GVL_HMI.bVisionImagePrepared := fbVisionManualImages.bPrepared;
GVL_HMI.bVisionImage1Allowed := bVisionPbupKnown AND NOT bVisionPbupFitted;
IF NOT GVL_HMI.bVisionImage1Allowed AND (GVL_HMI.udiCameraManualImageSelection = 1) THEN
    GVL_HMI.udiCameraManualImageSelection := 0;
END_IF
GVL_HMI.bVisionPbupFittedApplied := bVisionPbupFitted;
GVL_HMI.bVisionPbupReferenceKnown := bVisionPbupKnown;
GVL_HMI.uiVisionPbupNest := uiVisionPbupNest;
GVL_HMI.bVisionImagePrepareAllowed := bVisionImagePermit AND bVisionPbupKnown
    AND NOT fbVisionManualImages.bBusy AND NOT fbVisionManualImages.bFault
    AND (usiManualCameraStep = 0)
    AND (fbVisionManualImages.bActive OR stVisionStatus.bHome)
    AND NOT GVL_HMI.bCameraManualBusy AND GVL_HMI.bCameraConnected
    AND GVL_EtherCAT.stVSKeyenceCamera.bRunStatus
    AND (GVL_HMI.udiCameraManualImageSelection >= 1) AND (GVL_HMI.udiCameraManualImageSelection <= 4)
    AND ((GVL_HMI.udiCameraManualImageSelection <> 1) OR NOT bVisionPbupFitted);
GVL_HMI.bVisionImageReleaseAllowed := fbVisionManualImages.bPrepared
    AND NOT fbVisionManualImages.bPartHeld AND (usiManualCameraStep = 0);
GVL_HMI.bCameraManualReady := bManualCameraTransportReady AND fbVisionManualImages.bPrepared
    AND (GVL_HMI.udiCameraManualImageSelection = fbVisionManualImages.udiPreparedImage)
    AND bVisionPbupKnown AND ((GVL_HMI.udiCameraManualImageSelection <> 1) OR NOT bVisionPbupFitted);
GVL_HMI.bCameraManualReady := GVL_HMI.bCameraManualReady
    OR (bManualCameraRecoveryAllowed AND NOT bManualCameraRecoveryActive);
GVL_HMI.bCameraManualBusy := GVL_HMI.bCameraManualBusy OR fbVisionManualImages.bBusy;
IF fbVisionManualImages.bActive OR fbVisionManualImages.bFault
    OR ((eMachineState = E_MachineState.Manual) AND stCommand.bVisionManualEnable) THEN
    GVL_HMI.sCameraManualMessage := fbVisionManualImages.sMessage;
END_IF
// One actionable reason. Prepared geometry is independent of camera transport.
IF (eMachineState = E_MachineState.Manual) AND stCommand.bVisionManualEnable THEN
    IF NOT stInputs.stSafety.bSafetyOk THEN
        GVL_HMI.sCameraManualMessage := 'Vision blocked: safety not ready';
    ELSIF NOT stInputs.bMainDoorClosed OR NOT GVL_Safety.bAirSupplySafe THEN
        GVL_HMI.sCameraManualMessage := 'Vision blocked: close door / restore air';
    ELSIF bManualCameraRecoveryActive OR bManualCameraRecoveryFailed THEN
        GVL_HMI.sCameraManualMessage := sManualCameraRecoveryMessage;
    ELSIF fbVisionManualImages.bCameraWarning AND fbVisionManualImages.bBusy THEN
        GVL_HMI.sCameraManualMessage := fbVisionManualImages.sMessage;
    ELSIF bVisionCameraStartBlocked THEN
        GVL_HMI.sCameraManualMessage := 'Camera error - use Camera Reset or retry Trigger';
    ELSIF NOT GVL_HMI.bCameraConnected OR NOT GVL_EtherCAT.stVSKeyenceCamera.bRunStatus THEN
        GVL_HMI.sCameraManualMessage := 'Camera not connected / not in RUN';
    ELSIF stIndexStatus.bBusy OR stIndexStatus.bTwoHandRequired
        OR (stInputs.bTwoHandsSafe AND NOT fbVisionManualImages.bActive)
        OR NOT stInputs.bIndexReady OR NOT stInputs.bIndexLocked
        OR (stInputs.eIndexPosition = E_TablePosition.Unknown) THEN
        GVL_HMI.sCameraManualMessage := 'Wait for locked index; release two-hand';
    ELSIF bRejectChuteStopRequestLatched OR stCommand.bStop OR stCommand.bReset THEN
        GVL_HMI.sCameraManualMessage := 'Vision blocked: Stop/Reset active';
    ELSIF NOT stVisionNest.bPartPresent THEN
        GVL_HMI.sCameraManualMessage := 'No tracked product at Vision';
    ELSIF fbVisionManualImages.bFault OR fbVisionManualImages.bBusy THEN
        GVL_HMI.sCameraManualMessage := fbVisionManualImages.sMessage;
    ELSIF bVisionImageJogBusy OR bVisionManualSequenceActive OR bVisionManualHomeActive THEN
        GVL_HMI.sCameraManualMessage := 'Finish Vision jog / HOME / sequence first';
    ELSIF fbVisionManualImages.bCameraWarning THEN
        GVL_HMI.sCameraManualMessage := fbVisionManualImages.sMessage;
    ELSIF NOT bVisionPbupKnown THEN
        GVL_HMI.sCameraManualMessage := 'Confirm PBUP fitted state for this nest';
    ELSIF (GVL_HMI.udiCameraManualImageSelection < 1) OR (GVL_HMI.udiCameraManualImageSelection > 4) THEN
        GVL_HMI.sCameraManualMessage := 'Select an image';
    ELSIF (GVL_HMI.udiCameraManualImageSelection <> 1) AND NOT bVisionPbupFitted
        AND NOT stVisionNest.bLoadSetComplete THEN
        GVL_HMI.sCameraManualMessage := 'Mounting requires a complete paired load';
    ELSIF NOT fbVisionManualImages.bActive AND NOT stVisionStatus.bHome THEN
        GVL_HMI.sCameraManualMessage := 'Return Vision tooling HOME before Prepare';
    ELSIF bManualCameraDrainResult THEN
        GVL_HMI.sCameraManualMessage := 'Camera: clearing previous result handshake';
    ELSIF GVL_HMI.bCameraManualBusy THEN
        GVL_HMI.sCameraManualMessage := 'Camera: loading program / capture in progress';
    ELSIF fbVisionManualImages.bPrepared
        AND (GVL_HMI.udiCameraManualImageSelection = fbVisionManualImages.udiPreparedImage) THEN
        IF bManualCameraTransportReady THEN
            GVL_HMI.sCameraManualMessage := 'Position ready - press Camera Trigger';
        ELSE
            GVL_HMI.sCameraManualMessage := 'Position ready - waiting for camera handshake';
        END_IF
    ELSE
        GVL_HMI.sCameraManualMessage := 'Press Prepare Position for the selected image';
    END_IF
END_IF
GVL_HMI.sVisionPbupStatus := CONCAT('Nest ', UINT_TO_STRING(uiVisionPbupNest));
IF (uiVisionPbupNest < 1) OR (uiVisionPbupNest > 4) THEN
    GVL_HMI.sVisionPbupStatus := 'Wait for a known, locked index position';
ELSIF NOT stVisionNest.bPartPresent THEN
    GVL_HMI.sVisionPbupStatus := CONCAT(GVL_HMI.sVisionPbupStatus, ': no tracked part; load at operator station');
ELSIF NOT bVisionPbupKnown THEN
    GVL_HMI.sVisionPbupStatus := CONCAT(GVL_HMI.sVisionPbupStatus, ': confirm saved PBUP state');
ELSIF bVisionPbupFitted THEN
    GVL_HMI.sVisionPbupStatus := CONCAT(GVL_HMI.sVisionPbupStatus, ': PBUP fitted');
ELSE
    GVL_HMI.sVisionPbupStatus := CONCAT(GVL_HMI.sVisionPbupStatus, ': PBUP not fitted');
END_IF
IF stVisionNest.bPartPresent AND bVisionPbupKnown AND (uiVisionPbupNest >= 1) AND (uiVisionPbupNest <= 4) THEN
    IF aVisionPbupSource[uiVisionPbupNest] = 1 THEN
        GVL_HMI.sVisionPbupStatus := CONCAT(GVL_HMI.sVisionPbupStatus, ' / new paired load');
    ELSIF aVisionPbupSource[uiVisionPbupNest] = 2 THEN
        GVL_HMI.sVisionPbupStatus := CONCAT(GVL_HMI.sVisionPbupStatus, ' / operator confirmed');
    ELSE
        GVL_HMI.sVisionPbupStatus := CONCAT(GVL_HMI.sVisionPbupStatus, ' / mounting completed');
    END_IF
END_IF


// Native event grid is the single engineer-feedback presentation on this tab.
GVL_MASTER.bVisionManualCameraWarning := (eMachineState = E_MachineState.Manual)
    AND fbVisionManualImages.bCameraWarning;
GVL_MASTER.bVisionManualGridActive := (eMachineState = E_MachineState.Manual)
    AND stCommand.bVisionManualEnable;
GVL_MASTER.bVisionManualGridWarning := GVL_MASTER.bVisionManualGridActive
    AND NOT GVL_HMI.bCameraManualReady AND NOT GVL_HMI.bCameraManualBusy
    AND NOT fbVisionManualImages.bFault AND NOT fbVisionManualImages.bCameraWarning
    AND NOT bVisionCameraStartBlocked AND NOT bManualCameraRecoveryFailed;

// =====================================================
// VISION MANUAL MODE - HOME COMPLETION
// =====================================================

// Release Home ownership once FB_VisionStation has
// completed the controlled homing sequence and is Ready.
IF (eMachineState = E_MachineState.Manual)
    AND bVisionManualHomeActive
    AND fbVision.IsReady()
THEN
    bVisionManualHomeActive := FALSE;
END_IF;

// Release Home ownership if Vision enters Fault.
IF (eMachineState = E_MachineState.Manual)
    AND bVisionManualHomeActive
    AND fbVision.IsFaulted()
THEN
    bVisionManualHomeActive := FALSE;
END_IF;

// =====================================================
// VISION MANUAL MODE - RUN SEQUENCE COMPLETION
// =====================================================

// Complete manual Run Sequence.
// Return FB_VisionStation from Done to Ready.
IF (eMachineState = E_MachineState.Manual)
    AND bVisionManualSequenceActive
    AND fbVision.IsDone()
THEN
    fbVision.RequestReset();
    bVisionManualSequenceActive := FALSE;
END_IF;


// Abort manual Run Sequence ownership if Vision faults.
// The station fault remains available for the normal
// machine fault / diagnostic handling.
IF (eMachineState = E_MachineState.Manual)
    AND bVisionManualSequenceActive
    AND fbVision.IsFaulted()
THEN
    bVisionManualSequenceActive := FALSE;
END_IF;
// =====================================================
// VISION MANUAL MODE - OUTPUT OVERRIDE
// =====================================================
// Applied AFTER fbVision.Update() because FB_VisionStation owns these
// requests during Initialising / ReadyToStart / AutoCycle.
//
// Manual movement is accepted only when:
//   Manual Mode + Safety OK + Vision Manual Enable + movement permissive.
//
// Opposite requests are mutually interlocked here in the PLC.

// If Vision manual control is not enabled/allowed, do not permit any manual
// Vision motion request to survive into the physical output image.
IF (eMachineState = E_MachineState.Manual)
    AND NOT bVisionManualSequenceActive
    AND NOT bVisionManualHomeActive
    AND NOT fbVisionManualImages.bActive AND NOT bVisionImageOwnedBeforeUpdate
    AND NOT fbVisionManualImages.bFault
THEN

    // Start from a safe manual command image every scan.
    bVisionHorizontalBackRequest := FALSE;
    bVisionHorizontalFrontRequest := FALSE;
    bVisionVerticalUpRequest := FALSE;
    bVisionVerticalDownRequest := FALSE;

    bVisionGripCloseRequest := FALSE;
    bVisionGripOpenRequest := FALSE;
    bVisionRotate0Request := FALSE;
    bVisionRotate180Request := FALSE;



    // =====================================================
    // VISION MANUAL - COMMAND EDGES
    // =====================================================

    // Horizontal - KEEP EXACTLY AS VALIDATED
    rtVisionManualHorizontalBack(
        CLK := stCommand.bVisionHorizontalBackRequest
    );

    rtVisionManualHorizontalFront(
        CLK := stCommand.bVisionHorizontalFrontRequest
    );

//     // Vertical
//     rtVisionManualVerticalUp(
//         CLK := stCommand.bVisionVerticalUpRequest
//     );
// 
//     );
// 
//     rtVisionManualVerticalFullDown(
//         CLK := stCommand.bVisionVerticalFullDownRequest
//     );
// 
// 	rtVisionManualGripOpen(
// 		CLK := stCommand.bVisionGripOpenRequest
// 	);
// 	
// 	rtVisionManualGripClose(
// 		CLK := stCommand.bVisionGripCloseRequest
// 	);

    IF bVisionManualEnableAllowed
        AND stCommand.bVisionManualEnable
    THEN


        // =====================================================
        // VISION MANUAL - HORIZONTAL
        // =====================================================
        // KEEP EXACTLY AS VALIDATED.
        //
        // BACK = HOME

        tpVisionManualHorizontalBack(
            IN :=
                rtVisionManualHorizontalBack.Q
                AND bVisionHorizontalBackAllowed,
            PT := T#1S
        );

        // FRONT
        tpVisionManualHorizontalFront(
            IN :=
                rtVisionManualHorizontalFront.Q
                AND bVisionHorizontalFrontAllowed,
            PT := T#1S
        );

	

        // Never command both directions simultaneously.
        IF tpVisionManualHorizontalBack.Q
            AND NOT tpVisionManualHorizontalFront.Q
        THEN

            bVisionHorizontalBackRequest := TRUE;
            bVisionHorizontalFrontRequest := FALSE;

        ELSIF tpVisionManualHorizontalFront.Q
            AND NOT tpVisionManualHorizontalBack.Q
        THEN

            bVisionHorizontalFrontRequest := TRUE;
            bVisionHorizontalBackRequest := FALSE;

        END_IF;

		// =====================================================
		// VISION MANUAL - VERTICAL
		// =====================================================
		//
		// UP:
		//     Vertical UP until UP feedback.
		//
		// INTERMEDIATE:
		//     3. Drive Vertical DOWN.
		//     4. Stop command when cylinder leaves UP.
		//
		// FULL DOWN:
		//     3. Drive Vertical DOWN.
		//     4. Stop at full DOWN feedback.
		//
		// HMI commands are one-scan requests.
		// No timer is used.
		
		
		// -----------------------------------------------------
		// ACCEPT NEW TARGET
		// -----------------------------------------------------
		
        IF stCommand.bVisionVerticalUpRequest AND bVisionVerticalUpAllowed THEN
            bVisionManualVerticalUpActive := TRUE;
            bVisionManualVerticalFullDownActive := FALSE;
        ELSIF stCommand.bVisionVerticalFullDownRequest AND bVisionVerticalFullDownAllowed THEN
            bVisionManualVerticalUpActive := FALSE;
            bVisionManualVerticalFullDownActive := TRUE;
        END_IF
        IF bVisionManualVerticalUpActive THEN
            bVisionVerticalDownRequest := FALSE;
            bVisionVerticalUpRequest := NOT stInputs.bVerticalMiniSlideRetracted;
            IF stInputs.bVerticalMiniSlideRetracted THEN
                bVisionVerticalUpRequest := FALSE;
                bVisionManualVerticalUpActive := FALSE;
            END_IF
        ELSIF bVisionManualVerticalFullDownActive THEN
            bVisionVerticalUpRequest := FALSE;
            bVisionVerticalDownRequest := NOT stInputs.bVerticalMiniSlideExtended;
            IF stInputs.bVerticalMiniSlideExtended THEN
                bVisionVerticalDownRequest := FALSE;
                bVisionManualVerticalFullDownActive := FALSE;
            END_IF
        END_IF

		// =====================================================
		// VISION MANUAL - GRIP
		// =====================================================
		// Momentary command.
		// HMI request is converted to a one-scan PLC pulse in
		// PRG_HmiCommands.
		//
		// No timer is required.
		// OPEN and CLOSE are mutually exclusive.
		
		IF stCommand.bVisionGripOpenRequest
			AND NOT stCommand.bVisionGripCloseRequest
			AND bVisionGripOpenAllowed
		THEN
		
			bVisionGripOpenRequest := TRUE;
			bVisionGripCloseRequest := FALSE;
		
		ELSIF stCommand.bVisionGripCloseRequest
			AND NOT stCommand.bVisionGripOpenRequest
			AND bVisionGripCloseAllowed
		THEN
		
			bVisionGripOpenRequest := FALSE;
			bVisionGripCloseRequest := TRUE;
		
		ELSE
		
			bVisionGripOpenRequest := FALSE;
			bVisionGripCloseRequest := FALSE;
		
		END_IF


		// =====================================================
		// VISION MANUAL - ROTATION
		// =====================================================
		// HMI command is a one-scan request.
		// PLC keeps the output active until position feedback.
		// No timer is required.
		
		// Start 0Â°
		IF stCommand.bVisionRotate0Request
			AND bVisionRotate0Allowed
			AND NOT bVisionManualRotate180Active
		THEN
			bVisionManualRotate0Active := TRUE;
		END_IF
		
		// Start 180Â°
		IF stCommand.bVisionRotate180Request
			AND bVisionRotate180Allowed
			AND NOT bVisionManualRotate0Active
		THEN
			bVisionManualRotate180Active := TRUE;
		END_IF
		
		// Execute movement
		IF bVisionManualRotate0Active THEN
		
			bVisionRotate0Request := TRUE;
			bVisionRotate180Request := FALSE;
		
			IF bVisionRotate0Confirmed THEN
				bVisionRotate0Request := FALSE;
				bVisionManualRotate0Active := FALSE;
			END_IF
		
		ELSIF bVisionManualRotate180Active THEN
		
			bVisionRotate0Request := FALSE;
			bVisionRotate180Request := TRUE;
		
			IF bVisionRotate180Confirmed THEN
				bVisionRotate180Request := FALSE;
				bVisionManualRotate180Active := FALSE;
			END_IF
		
		ELSE
		
			bVisionRotate0Request := FALSE;
			bVisionRotate180Request := FALSE;
		
		END_IF


	ELSE
	
		// Vision Manual Enable removed:
		// cancel unfinished manual movements.

		bVisionManualVerticalUpActive := FALSE;
		bVisionManualVerticalFullDownActive := FALSE;
		bVisionManualRotate0Active := FALSE;
		bVisionManualRotate180Active := FALSE;
	
	END_IF

ELSE

    // Leaving Manual also cancels unfinished manual sequences.
    bVisionManualVerticalUpActive := FALSE;

    bVisionManualVerticalFullDownActive := FALSE;

    bVisionManualRotate0Active := FALSE;
    bVisionManualRotate180Active := FALSE;

END_IF

stVisionStatus.bFault := stVisionStatus.bFault OR fbVisionManualImages.bFault;
IF fbVisionManualImages.bActive OR fbVisionManualImages.bFault THEN
    stVisionStatus.sDiagnostic := fbVisionManualImages.sMessage;
END_IF

// Current station/nest status for HMI.
stPatchDispenseStatus.bPartPresent := bPatchDispenseRequired;
stHeatStakeStatus.bPartPresent := bHeatStakeRequired;
stVisionStatus.bPartPresent := bVisionRequired;

// Homing is an internal machine-initialisation activity, not an automatic
// process cycle. Keep FB_VisionStation.IsBusy() unchanged for controlled-stop
// logic, but do not publish Vision as Busy to the operator while the machine is
// in System Initialising.
IF eMachineState = E_MachineState.Initialising THEN
    stVisionStatus.bBusy := FALSE;
END_IF

// Manual indication follows current HOME feedback, independently of the station FB state.
// Individual manual movements are owned by the machine and can leave the station FB idle.
IF eMachineState = E_MachineState.Manual THEN
    stVisionStatus.bBusy :=
        NOT stVisionStatus.bHome
        OR bVisionManualSequenceActive
        OR bVisionManualHomeActive
        OR fbVisionManualImages.bActive;

    stVisionStatus.bReady :=
        stVisionStatus.bHome
        AND NOT stVisionStatus.bBusy
        AND bVisionManualEnableAllowed
        AND stCommand.bVisionManualEnable
        AND NOT fbVision.IsFaulted() AND NOT fbVisionManualImages.bFault;
END_IF

// "Ready" on the Heat Stake HMI is an operational indication, not an
// Initialising indication.
//
// FB_HeatStakeStation is intentionally enabled during System Initialising so
// it can establish/check its safe initial position. Its internal IsReady()
// state is still allowed to become TRUE there, because machine Initialising
// may depend on it. Only the published HMI Ready indication is gated.
//
// Show Ready only in states where an engineer/operator can actually use the
// station.
stHeatStakeStatus.bReady :=
    stHeatStakeStatus.bReady
    AND (
        (eMachineState = E_MachineState.ReadyToStart)
        OR (eMachineState = E_MachineState.AutoCycle)
        OR (eMachineState = E_MachineState.Manual)
    );

IF NOT bPatchDispenseRequired THEN
    stPatchDispenseStatus.eResultStatus := E_StationResultStatus.NotTested;
ELSIF stPatchDispenseNest.stPatchDispenseResult.bValid THEN
    IF stPatchDispenseNest.stPatchDispenseResult.bPassed THEN
        stPatchDispenseStatus.eResultStatus := E_StationResultStatus.Pass;
    ELSE
        stPatchDispenseStatus.eResultStatus := E_StationResultStatus.Fail;
    END_IF
ELSE
    stPatchDispenseStatus.eResultStatus := E_StationResultStatus.NotTested;
END_IF

IF stHeatStakeNest.stHeatStakeResult.bValid
    AND (stHeatStakeNest.stHeatStakeResult.udiAlertCode = GVL_MASTER.udiHeatStakePatchMissingAlertCode) THEN
    stHeatStakeStatus.eResultStatus := E_StationResultStatus.Fail;
ELSIF NOT bHeatStakeRequired THEN
    stHeatStakeStatus.eResultStatus := E_StationResultStatus.NotTested;
ELSIF stHeatStakeNest.stHeatStakeResult.bValid THEN
    IF stHeatStakeNest.stHeatStakeResult.bPassed THEN
        stHeatStakeStatus.eResultStatus := E_StationResultStatus.Pass;
    ELSE
        stHeatStakeStatus.eResultStatus := E_StationResultStatus.Fail;
    END_IF
ELSE
    stHeatStakeStatus.eResultStatus := E_StationResultStatus.NotTested;
END_IF

IF NOT bVisionRequired THEN
    stVisionStatus.eResultStatus := E_StationResultStatus.NotTested;
ELSIF stVisionNest.stVisionResult.bValid THEN
    IF stVisionNest.stVisionResult.bPassed THEN
        stVisionStatus.eResultStatus := E_StationResultStatus.Pass;
    ELSE
        stVisionStatus.eResultStatus := E_StationResultStatus.Fail;
    END_IF
ELSE
    stVisionStatus.eResultStatus := E_StationResultStatus.NotTested;
END_IF

bAllRequiredStationsReady :=
    ((NOT bPatchDispenseRequired) OR fbPatchDispense.IsReady())
    AND ((NOT bHeatStakeRequired) OR fbHeatStake.IsReady())
    AND ((NOT bVisionRequired) OR fbVision.IsReady());

bAllRequiredStationsComplete :=
    ((NOT bPatchDispenseRequired) OR fbPatchDispense.IsDone())
    AND ((NOT bHeatStakeRequired) OR fbHeatStake.IsDone())
    AND ((NOT bVisionRequired) OR fbVision.IsDone());

// TRUE from support extension through the simulated process and support
// retraction of at least one active station.
bAnyStationInProcess :=
    fbPatchDispense.IsBusy()
    OR fbHeatStake.IsBusy()
    OR fbVision.IsBusy();

IF (eProcessCycleState = E_CycleState.WaitingForProcessesComplete)
    AND bAllRequiredStationsComplete
    AND NOT bCycleResultsStored
THEN

	IF bPatchDispenseRequired THEN
	
		// Capture the station result once.
		stPatchDispenseCycleResult := fbPatchDispense.GetResult();
	
		// Store the Patch Dispense result in the physical nest.
		fbNestManager.StorePatchDispenseResultAtPosition(
			ePosition := stConfig.ePatchDispensePosition,
			stResult := stPatchDispenseCycleResult
		);
	
		IF stPatchDispenseCycleResult.bValid AND NOT stPatchDispenseCycleResult.bPassed THEN
			FinaliseAndRecordAtPosition(stConfig.ePatchDispensePosition);
		END_IF

	END_IF

    IF bHeatStakeRequired THEN
        stHeatStakeCycleResult := fbHeatStake.GetResult();
        fbNestManager.StoreHeatStakeResultAtPosition(
            ePosition := stConfig.eHeatStakePosition,
            stResult := stHeatStakeCycleResult
        );
        IF stHeatStakeCycleResult.bValid AND NOT stHeatStakeCycleResult.bPassed THEN
            FinaliseAndRecordAtPosition(stConfig.eHeatStakePosition);
        END_IF
    END_IF

    IF bVisionRequired THEN
        fbNestManager.StoreVisionResultAtPosition(
            ePosition := stConfig.eVisionPosition,
            stResult := fbVision.GetResult()
        );
    END_IF
	
    FinaliseAndRecordAtPosition(stConfig.eVisionPosition);

// Prevent this cycle result from being stored/finalised again.
bCycleResultsStored := TRUE;


END_IF

// =====================================================
// REPROCESS POPUP - OPERATOR STATION
// =====================================================
// 
// Activate Reprocess requirement when a Reprocess
// part is present at the Operator Station.
IF (stOperatorNest.ePosition = E_TablePosition.Position1)
    AND (stOperatorNest.eDisposition = E_PartDisposition.Reprocess)
    AND stOperatorNest.bPartPresent
THEN
    bReprocessAcknowledgePending := TRUE;
END_IF

// Reset acknowledgement memory only when there is
// no active Reprocess acknowledgement pending
// and the operator nest is empty.
IF NOT stOperatorNest.bPartPresent
    AND NOT bReprocessAcknowledgePending
THEN
    bReprocessPopupAcknowledged := FALSE;
END_IF

// Acknowledge the current Reprocess part.
IF GVL_HMI.stCommands.bReprocessPopupAcknowledge THEN
    bReprocessPopupAcknowledged := TRUE;
    bReprocessAcknowledgePending := FALSE;
    GVL_HMI.stCommands.bReprocessPopupAcknowledge := FALSE;
END_IF

// // Require acknowledgement only for an unacknowledged
// // Reprocess part physically present at the Operator Station.
// IF (stOperatorNest.ePosition = E_TablePosition.Position1)
//     AND (stOperatorNest.eDisposition = E_PartDisposition.Reprocess)
//     AND stOperatorNest.bPartPresent
//     AND NOT bReprocessPopupAcknowledged
// THEN
//     bReprocessAcknowledgePending := TRUE;
// END_IF

// Popup remains requested until acknowledged,
// // even if the part is physically removed.
// GVL_HMI.stStatus.bReprocessPopupRequest :=
//     bReprocessAcknowledgePending;
// Reprocess popup request.
// Keep the PLC interlock independent from popup visibility.

rtReprocessIndexAttempt(
    CLK := stInputs.bTwoHandsSafe
);

// Generate a new FALSE -> TRUE transition when the
// operator attempts to index with Reprocess pending.
IF NOT bReprocessAcknowledgePending THEN

    GVL_HMI.stStatus.bReprocessPopupRequest := FALSE;

ELSIF rtReprocessIndexAttempt.Q THEN

    GVL_HMI.stStatus.bReprocessPopupRequest := FALSE;

ELSE

    GVL_HMI.stStatus.bReprocessPopupRequest := TRUE;

END_IF
// Request popup only for an unacknowledged Reprocess part
// physically present at the Operator Station.
// GVL_HMI.stStatus.bReprocessPopupRequest :=
//     (stOperatorNest.ePosition = E_TablePosition.Position1)
//     AND (stOperatorNest.eDisposition = E_PartDisposition.Reprocess)
//     AND stOperatorNest.bPartPresent
//     AND NOT bReprocessPopupAcknowledged;

// Clear an old processed record only after operator disposition is complete.
// A newly loaded part is not cleared because its load edge has already reset
// stResult.bValid to FALSE in FB_NestTableManager.
IF stOperatorStatus.bExchangeComplete
    AND (
        stOperatorNest.stResult.bValid
        OR (stOperatorNest.eDisposition = E_PartDisposition.Reprocess)
    )
    AND NOT stInputs.bLoadingStationEaglePresent
    AND NOT stInputs.bLoadingStationPbupPresent
THEN

    fbNestManager.ClearOperatorNest(
        stConfig.eOperatorPosition
    );

END_IF




stOutputsInternal.bStation1SupportExtend := FALSE; // Removed Station 1 nest support.
stOutputsInternal.bStation1SupportRetract := FALSE; // Reserved compatibility output.
stOutputsInternal.bStation2SupportExtend := bStation2SupportExtendRequest;
stOutputsInternal.bStation2SupportRetract := bStation2SupportRetractRequest;
stOutputsInternal.bStation3SupportExtend := FALSE; // Removed hardware.
stOutputsInternal.bStation3SupportRetract := FALSE; // Removed hardware.
stOutputsInternal.bVisionHorizontalBack := bVisionHorizontalBackRequest;
stOutputsInternal.bVisionHorizontalFront := bVisionHorizontalFrontRequest;
stOutputsInternal.bVisionVerticalUp := bVisionVerticalUpRequest;
stOutputsInternal.bVisionVerticalDown := bVisionVerticalDownRequest;
stOutputsInternal.bVisionLimitOff := FALSE; // Removed hardware.
stOutputsInternal.bVisionLimitOn := FALSE; // Removed hardware.
stOutputsInternal.bVisionGripClose := bVisionGripCloseRequest;
stOutputsInternal.bVisionGripOpen := bVisionGripOpenRequest;
stOutputsInternal.bVisionRotate0 := bVisionRotate0Request;
stOutputsInternal.bVisionRotate180 := bVisionRotate180Request;
stOutputsInternal.bHeatStakeHeadLock := bHeatStakeHeadLockRequest;
stOutputsInternal.bHeatStakeHeadUnlock := bHeatStakeHeadUnlockRequest;
stOutputsInternal.bHeatStakeHeadDown := bHeatStakeHeadDownRequest;
stOutputsInternal.bHeatStakeHeadUp := bHeatStakeHeadUpRequest;
stPermissives.bAirSupplyReady := GVL_Safety.bAirSupplySafe;


// Patch actuator ownership: HOME/sequence, individual Manual actions, then index hold-UP.
bPatchHoldUpAllowed := bPatchDispenseCommissioned AND stInputs.stSafety.bSafetyOk
    AND stInputs.bMainDoorClosed AND GVL_Safety.bAirSupplySafe
    AND ((eMachineState = E_MachineState.AutoCycle)
        OR ((eMachineState = E_MachineState.Manual)
            AND NOT bPatchManualVerticalDownHeld AND NOT stPatchDispenseStatus.bFault)
        OR ((eMachineState = E_MachineState.Stopping) AND stIndexStatus.bBusy));
stOutputsInternal.bPatchVerticalUp := FALSE;
stOutputsInternal.bPatchVerticalDown := FALSE;
stOutputsInternal.bPatchDispenserAir := FALSE;
IF stInputs.stSafety.bSafetyOk AND stInputs.bMainDoorClosed
    AND GVL_Safety.bAirSupplySafe AND bPatchDispenseCommissioned THEN
    IF fbPatchDispense.IsBusy() OR (eMachineState = E_MachineState.Initialising) THEN
        stOutputsInternal.bPatchVerticalDown := bPatchSequenceDownRequest;
        stOutputsInternal.bPatchVerticalUp := bPatchHomeVerticalUpRequest
            AND NOT bPatchSequenceDownRequest;
        stOutputsInternal.bPatchDispenserAir := bPatchSequenceAirRequest;
    ELSIF bPatchManualAllowed THEN
        stOutputsInternal.bPatchVerticalDown := bPatchManualVerticalDownHeld
            AND NOT stCommand.bIndexerManualEnable;
        stOutputsInternal.bPatchVerticalUp := bPatchManualVerticalUpHeld
            AND NOT stOutputsInternal.bPatchVerticalDown;
        stOutputsInternal.bPatchDispenserAir := tpPatchAirBlow.Q;
    ELSE
        stOutputsInternal.bPatchVerticalUp := bPatchHoldUpAllowed;
    END_IF
END_IF

// Same criterion used by the validated Silicone Station:
// the machine waits until the door supervisor confirms automatic readiness.
stPermissives.bDoorInitialisationReady :=
    NOT fbMainDoorLock.IsFaulted()
    AND fbMainDoorLock.IsReadyForAutomatic();
stPermissives.bIndexInitialisationReady := NOT fbIndex.IsFaulted();
// Heat Stake is the only fitted nest support. Require its real retracted
// feedback and reject contradictory feedback. Patch transfer vertical and
// all other index permissives remain separate below.
stPermissives.bStationsHome :=
    stInputs.bStation2SupportRetracted
    AND NOT stInputs.bStation2SupportExtended;

stPermissives.bInitialisationAllowed := stInputs.stSafety.bSafetyOk
    AND stPermissives.bAirSupplyReady
    AND stPermissives.bDoorInitialisationReady
    AND stPermissives.bIndexInitialisationReady;

stPermissives.bSafetyIndexPermissive := stInputs.stSafety.bMotionSafetyPermitted;

stPermissives.bOperatorIndexPermissive :=
    stOperatorStatus.bIndexPermissive
    AND bOperatorLoadValid
    AND NOT bReprocessAcknowledgePending;

stPermissives.bStationsIndexPermissive := stPermissives.bStationsHome
    AND bPatchVerticalIndexReady
    AND (GVL_Motion.stPatchFeedSettings.bUsePatchVerticalFeedback
        OR stOutputsInternal.bPatchVerticalUp)
    AND NOT fbPatchDispense.IsBusy() AND NOT fbPatchFeedManager.stStatus.bDriveBusy
    AND NOT bPatchManualVerticalDownHeld
    AND NOT stOutputsInternal.bPatchVerticalDown
    AND NOT fbVisionManualImages.bActive AND NOT bVisionImageRecoveryRequired
    AND ((eMachineState <> E_MachineState.Manual)
        OR (stVisionStatus.bHome AND bHeatStakeManualHomePosition AND NOT fbVisionManualImages.bFault
            AND NOT bVisionImageJogBusy AND NOT bVisionManualHomeActive AND NOT bVisionManualSequenceActive
            AND NOT bManualCameraRecoveryActive));
// IMPORTANT:
// The operator exchange permissive is a START permissive only.
// Once the table starts moving, FB_OperatorStation intentionally leaves
// ExchangeComplete and bOperatorIndexPermissive becomes FALSE.
// Therefore it must NOT be part of the continuous movement permissive passed
// to FB_IndexTable4, otherwise the index faults immediately with
// MovementPermissiveLost as soon as motion begins.
//
// ProcessCycle still checks bOperatorIndexPermissive BEFORE RequestMove().
stPermissives.bIndexMoveAllowed :=
    stPermissives.bSafetyIndexPermissive
    AND stPermissives.bStationsIndexPermissive;
	
fbCommissioningGuard.Cyclic(bDispenseCommissioned := bPatchDispenseCommissioned, 
bHeatStakeCommissioned := bHeatStakeCommissioned, 
bVisionCommissioned := bVisionCommissioned,
bCoreCommissioningMode := bCoreCommissioningMode, 
bCoreReady := ((eMachineState = E_MachineState.ReadyToStart) 
				OR (eMachineState = E_MachineState.Dwell)
				OR (eMachineState = E_MachineState.AutoCycle)), 
bAutoCycleAllowed => bAutoCycleAllowed, 
sBlockReason => sAutoCycleBlockReason);

// Camera RUN is an independent automatic-operation requirement.
// Commissioning mode must not bypass this camera prerequisite.
IF NOT GVL_EtherCAT.stVSKeyenceCamera.bRunStatus THEN
    bAutoCycleAllowed := FALSE;
    sAutoCycleBlockReason := 'Vision camera not in RUN - select RUN in VS Creator';
ELSIF bVisionCameraStartBlocked THEN
    bAutoCycleAllowed := FALSE;
    sAutoCycleBlockReason := 'Vision camera error - follow camera recovery procedure before Start';
END_IF

stPermissives.bAutoCycleAllowed := bAutoCycleAllowed;

fbProcessCycle.Cyclic(
    bEnable := (eMachineState = E_MachineState.AutoCycle),
    bResetRequest := stCommand.bReset,
    bStopRequest :=
        stCommand.bStop
        OR stInputs.bEventCycleStopRequest
        OR bRejectChuteStopRequestLatched
        OR NOT GVL_EtherCAT.stVSKeyenceCamera.bRunStatus,
    bTwoHandsSafe := stInputs.bTwoHandsSafe,
    bSafetyOk := stInputs.stSafety.bSafetyOk,
    bIndexReady := stInputs.bIndexReady,
    bIndexLocked := stInputs.bIndexLocked,
    bIndexBusy := stIndexStatus.bBusy,
    bIndexFaulted := fbIndex.IsFaulted(),
	bHeaterDwellPending := bHeaterDwellRequestLatched,
    bStationsIndexPermissive := stPermissives.bStationsIndexPermissive,
    bOperatorIndexPermissive := stPermissives.bOperatorIndexPermissive,
    bTemperatureIndexPermissive := stHeatStakeTemperatureStatus.bIndexTemperatureReady,
    bNestEnableIndexPermissive := NOT bDisabledNestPartPresent,
    bAllStationsReady := bAllRequiredStationsReady,
    bAllStationsComplete := bAllRequiredStationsComplete,
    bAnyStationFault :=
        fbPatchDispense.IsFaulted()
        OR fbHeatStake.IsFaulted()
        OR fbVision.IsFaulted(),
    tSequenceTimeout := UDINT_TO_TIME(
        UINT_TO_UDINT(LIMIT(UINT#1, GVL_Persistent.uiAutoCycleIdleTimeoutMin, UINT#1440)) * UDINT#60000),
    bStartStations => bProcessStartStations,
    bStopStations => bProcessStopStations,
    bRequestIndex => bProcessRequestIndex,
    bCycleActive => bProcessCycleActive,
    bCompletePulse => bProcessCycleCompletePulse,
    bFault => bProcessCycleFault,
    bSequenceTimeoutFault => bProcessCycleTimeoutFault,
    bStopPendingStatus => bProcessStopPending,
    bAutomaticStopRequest => bProcessAutomaticStopRequest,
    bDisabledNestIndexAttempt => bDisabledNestIndexAttempt,
    eState => eProcessCycleState
);

// Stop Request is latched immediately so the operator request is never lost,
// even when an automatic station process is still running.
//
// Sources:
// - physical/HMI Stop command;
// - existing Events-cycle Stop Request;
// - Configured automatic inactivity request from FB_ProcessCycle.
//
// The existing Events/DataGrid logic is intentionally untouched, so the
// operator Stop Request indication continues to appear immediately as before.
IF (eMachineState = E_MachineState.AutoCycle)
    AND (
        stCommand.bStop
        OR stInputs.bEventCycleStopRequest
        OR bProcessAutomaticStopRequest
        OR bRejectChuteStopRequestLatched
        OR NOT GVL_EtherCAT.stVSKeyenceCamera.bRunStatus
    )
THEN
    bAutoCycleStopRequestLatched := TRUE;
END_IF

IF bDisabledNestIndexAttempt AND bDisabledNestPartPresent THEN
    bDisabledNestPartPopupRequest := TRUE;
    uiDisabledNestPartPopupNestId := uiDisabledNestPartNestId;
END_IF

// Popup OK only closes the request. If the part is still present, the next
// fresh index attempt requests the popup again.
IF stCommand.bAcknowledgeDisabledNestPartPopup THEN
    bDisabledNestPartPopupRequest := FALSE;
END_IF

// Block only a NEW automatic index request; preserve in-progress motion permissives.
IF bProcessRequestIndex AND GVL_EtherCAT.stVSKeyenceCamera.bRunStatus
    AND bOperatorLoadValid AND stPermissives.bOperatorIndexPermissive
    AND stInputs.bTwoHandsSafe AND stInputs.bIndexReady AND stInputs.bIndexLocked
    AND NOT stIndexStatus.bBusy AND (stInputs.eIndexPosition <> E_TablePosition.Unknown) THEN
    bIndexMoveAccepted := fbIndex.RequestMove();
END_IF



// =========================================================
// HMI HEARTBEAT MONITORING
// =========================================================
tonHMIAliveOn(
    IN := GVL_HMI.bHMIAlive,
    PT := T#2S
);

tonHMIAliveOff(
    IN := NOT GVL_HMI.bHMIAlive,
    PT := T#2S
);

bOutHMI := tonHMIAliveOn.Q OR tonHMIAliveOff.Q;


// =========================================================
// HMI UNAVAILABLE - STOPPED MESSAGE
// =========================================================

// Show the HMI unavailable message only while
// the machine is Stopped and heartbeat is missing.
GVL_HMI.bHmiLogoutStopped := bOutHMI AND (eMachineState = E_MachineState.Stopped);

// =========================================================
// HMI CONNECTION LOSS - SAFETY DROP REQUEST
// =========================================================
// A confirmed heartbeat timeout during an active machine
// state requests a TwinSAFE Run/Stop drop.
//
// Stopped and Stopping do not generate a new fault.

IF bOutHMI AND (
    (eMachineState = E_MachineState.Initialising)
    OR (eMachineState = E_MachineState.ReadyToStart)
    OR (eMachineState = E_MachineState.AutoCycle)
    OR (eMachineState = E_MachineState.Manual)
	OR (eMachineState = E_MachineState.Dwell)
) THEN
    bSafetyDropRequest := TRUE;
    // Preserve the trip reason through the existing HMI event/reset path.
    GVL_HMI.bHmiLogoutAutoCycle := TRUE;
END_IF

// =========================================================
// UNEXPECTED HMI LOGOUT
// =========================================================
// Logout is permitted in Stopped and Stopping.
// During operation, logout causes a machine Fault.
// Do not request a TwinSAFE run drop for a user-session event.

IF bLogoutHMI AND (
    (eMachineState = E_MachineState.Initialising)
    OR (eMachineState = E_MachineState.ReadyToStart)
    OR (eMachineState = E_MachineState.AutoCycle)
    OR (eMachineState = E_MachineState.Manual)
	OR (eMachineState = E_MachineState.Dwell)
) THEN
    GVL_HMI.bLogoutFaultActive := TRUE;
    bSafetyDropRequest := TRUE;
	GVL_HMI.bHmiLogoutAutoCycle := TRUE;
	GVL_HMI.bHmiLogoutStopped := FALSE;
END_IF

// TwinSAFE safety loss always places the machine in Fault, but it must NOT
// generate a PLC Run/Stop drop request. RunRequest must return TRUE so
// TwinSAFE can execute again and restore Safety_OK after the safety condition
// has recovered.
IF NOT stInputs.stSafety.bSafetyOk THEN
    eMachineState := E_MachineState.Fault;
END_IF

// PLC-originated immediate faults request a controlled TwinSAFE run drop.
// stInputs.bEventFault is the aggregate of active Events with bFault = TRUE.
// Re-check after component cyclic execution so a fault detected in this scan
// drops TwinSAFE immediately rather than waiting for the following PLC scan.
// Existing event/process-cycle faults are allowed during Initialising so the
// machine can restore pneumatic tooling to HOME.
IF (
        stInputs.bEventFault
        AND (eMachineState <> E_MachineState.Initialising)
    )
    OR fbIndex.IsFaulted()
    OR fbMainDoorLock.IsFaulted()
    OR (
        bProcessCycleFault
        AND (eMachineState <> E_MachineState.Initialising)
    )
    OR stHeatStakeTemperatureStatus.bFault
    OR bInitialisationTimeoutFault
    OR bStoppingTimeoutFault
THEN
    bSafetyDropRequest := TRUE;
    eMachineState := E_MachineState.Fault;
END_IF



CASE eMachineState OF
E_MachineState.PowerUp:
    bAutoCycleStopRequestLatched := FALSE;

    // Same lifecycle used by the validated Silicone Station core:
    // always enter a controlled stop before waiting for Reset.
    tonInitialising(IN := FALSE);
    tonStopping(IN := FALSE);
    eMachineState := E_MachineState.Stopping;

E_MachineState.Stopping:
    // Preserve an already-established pneumatic supply while stopping, but
    // never create a new air request here.
    //
    // Typical Stop path:
    // Ready/Auto/Manual (air latched) -> Stopping -> Stopped
    // Air remains ON while the door stays closed.
    //
    // Fault recovery / PowerUp path:
    // latch is FALSE -> Stopping remains depressurised.
    stOutputsInternal.bAirSupplyEnable :=
        bAirSupplyLatched AND stInputs.bMainDoorClosed;

    tonInitialising(IN := FALSE);
    tonStopping(IN := stIndexStatus.bBusy OR fbPatchFeedManager.stStatus.bBusy, PT := stConfig.tStoppingTimeout);
    bStoppingTimeoutFault := tonStopping.Q;
    IF bStoppingTimeoutFault THEN
        bSafetyDropRequest := TRUE;
        eMachineState := E_MachineState.Fault;
	// The removed Station 1 support no longer gates completion of Stopping.
	ELSIF NOT stIndexStatus.bBusy
        AND NOT fbPatchFeedManager.stStatus.bBusy
	THEN
		eMachineState := E_MachineState.Stopped;
	END_IF

E_MachineState.Stopped:
    bAutoCycleStopRequestLatched := FALSE;

    // Stopped never turns the air ON by itself.
    // It only preserves air that was previously latched by Initialising.
    // As soon as the main door opens, the global door-open rule clears the
    // latch and the ASU drops. Closing the door again does not restore it.
    stOutputsInternal.bAirSupplyEnable :=
        bAirSupplyLatched AND stInputs.bMainDoorClosed;

    tonInitialising(IN := FALSE);
    tonStopping(IN := FALSE);

    // The controlled Stop Request remains latched until Stopped is reached.
    // It is released only after the reject chute interlock was correctly
    // cleared by EMPTY + fresh Acknowledge.
    IF NOT bRejectChuteFullLatched THEN
        bRejectChuteStopRequestLatched := FALSE;
    END_IF

    IF stCommand.bReset
        AND stInputs.stSafety.bSafetyOk
        AND NOT bRejectChuteFullLatched
    THEN
        // Same recovery used by the Silicone Station: clear any stale
        // door-supervisor fault/state before automatic locking starts.
        fbMainDoorLock.Initialise();
        eMachineState := E_MachineState.Initialising;
    END_IF

E_MachineState.Initialising:
    // Only Initialising may establish the pneumatic-supply latch.
    IF stInputs.bMainDoorClosed THEN
        bAirSupplyLatched := TRUE;
    END_IF

    stOutputsInternal.bAirSupplyEnable := bAirSupplyLatched AND stInputs.bMainDoorClosed;
    tonStopping(IN := FALSE);

    // All commissioned stations must complete their HOME sequences.
    tonInitialising(
        IN := NOT (
            stPermissives.bInitialisationAllowed
            AND (usiHeatStakeManualActionStep = 0)
            AND stInputs.bHeatStakeHeadUp
            AND NOT stInputs.bHeatStakeHeadDown
            AND NOT bHeatStakeManualHeadUpTimeoutFault
            AND NOT bHeatStakeManualHeadDownTimeoutFault
            AND NOT bHeatStakeStationHeadSensorConflictFault
            AND ((NOT bVisionCommissioned) OR fbVision.IsReady())
            AND ((NOT bPatchDispenseCommissioned) OR fbPatchDispense.IsHome())
        ),
        PT := stConfig.tInitialiseTimeout
    );

    bInitialisationTimeoutFault := tonInitialising.Q;

    IF bInitialisationTimeoutFault THEN
        bSafetyDropRequest := TRUE;
        eMachineState := E_MachineState.Fault;
    ELSIF stPermissives.bInitialisationAllowed
        AND (usiHeatStakeManualActionStep = 0)
        AND stInputs.bHeatStakeHeadUp
        AND NOT stInputs.bHeatStakeHeadDown
        AND NOT bHeatStakeManualHeadUpTimeoutFault
        AND NOT bHeatStakeManualHeadDownTimeoutFault
        AND NOT bHeatStakeStationHeadSensorConflictFault
        //AND ((NOT bVisionCommissioned) OR fbVision.IsReady())
        AND ((NOT bPatchDispenseCommissioned) OR fbPatchDispense.IsHome())
    THEN
        tonInitialising(IN := FALSE);
        eMachineState := E_MachineState.ReadyToStart;
    END_IF

E_MachineState.ReadyToStart:
    stOutputsInternal.bAirSupplyEnable :=
        bAirSupplyLatched AND stInputs.bMainDoorClosed;

    IF bRejectChuteStopRequestLatched THEN
        eMachineState := E_MachineState.Stopping;

    ELSIF stCommand.bStop THEN
        eMachineState := E_MachineState.Stopping;

    ELSIF stCommand.bManualRequest
        AND stInputs.stSafety.bSafetyOk
        AND NOT stIndexStatus.bBusy
        AND NOT fbIndex.IsFaulted()
    THEN
        eMachineState := E_MachineState.Manual;
    ELSIF stCommand.bStart AND bAutoCycleAllowed AND fbMainDoorLock.IsReadyForAutomatic() THEN
		  IF stHeatStakeTemperatureStatus.bIndexTemperatureReady THEN
				// Heater is ready: start automatic operation.
				eMachineState := E_MachineState.AutoCycle;
			ELSE
				// Heater is below the operating temperature:
				// wait in Dwell before starting automatic operation.
				eMachineState := E_MachineState.Dwell;
			END_IF
	END_IF
	
	
E_MachineState.Dwell:

    // Keep pneumatic supply enabled while waiting for heater temperature.
    stOutputsInternal.bAirSupplyEnable :=
        bAirSupplyLatched AND stInputs.bMainDoorClosed;

    // Stop has priority over temperature recovery.
    IF bRejectChuteStopRequestLatched
        OR stCommand.bStop
        OR stInputs.bEventCycleStopRequest
        OR NOT GVL_EtherCAT.stVSKeyenceCamera.bRunStatus
    THEN
        eMachineState := E_MachineState.Stopping;

    ELSIF stHeatStakeTemperatureStatus.bIndexTemperatureReady
        AND bAutoCycleAllowed
        AND fbMainDoorLock.IsReadyForAutomatic()
        AND stInputs.stSafety.bSafetyOk
    THEN
        // Automatically resume AutoCycle when the heater is ready.
        eMachineState := E_MachineState.AutoCycle;
    END_IF
	

E_MachineState.AutoCycle:
    stOutputsInternal.bAirSupplyEnable :=
        bAirSupplyLatched AND stInputs.bMainDoorClosed;
		
		// =====================================================
		// HEATER DWELL - CONTROLLED TRANSITION
		// =====================================================
		// Wait until the current production cycle has finished,
		// all stations are idle and the index is stationary.
		
		IF bHeaterDwellRequestLatched
			AND NOT bAutoCycleStopRequestLatched
			AND (eProcessCycleState = E_CycleState.WaitingForProcessCycleTrigger)
			AND NOT bAnyStationInProcess
			AND NOT stIndexStatus.bBusy
			AND stInputs.bIndexReady
			AND stInputs.bIndexLocked
			AND stPermissives.bStationsIndexPermissive
			AND NOT bProcessStartStations
			AND NOT bProcessRequestIndex
		THEN
			bHeaterDwellRequestLatched := FALSE;
			eMachineState := E_MachineState.Dwell;
		END_IF

    // Stop Request is controlled, but ONLY an active process at one of the
    // three process stations is allowed to delay leaving AutoCycle.
    //
    // Heat Stake warm-up / temperature control is NOT a process and must not
    // hold the machine in AutoCycle after Stop Request.
    //
    // Likewise, the ProcessCycle coordinator state and index busy state do not
    // block the AutoCycle -> Stopping transition:
    // - ProcessCycle is disabled as soon as AutoCycle is left;
    // - if the index is already moving, the normal Stopping state waits for
    //   stIndexStatus.bBusy to clear before entering Stopped.
    //
    // Therefore the only controlled-stop hold condition here is:
    //     fbPatchDispense.IsBusy()
    //     OR fbHeatStake.IsBusy()
    //     OR fbVision.IsBusy()
    IF bAutoCycleStopRequestLatched
        AND NOT bAnyStationInProcess
    THEN
        bAutoCycleStopRequestLatched := FALSE;
        eMachineState := E_MachineState.Stopping;
    END_IF

E_MachineState.Manual:
    stOutputsInternal.bAirSupplyEnable :=
        bAirSupplyLatched AND stInputs.bMainDoorClosed;

    // Reject chute full = controlled stop in Manual Mode.
    // No new manual actions are accepted. Existing actions complete first.
    bManualRejectStopReady :=
        NOT bHeatStakeManualActionBusy
        AND NOT bHeatStakeManualStakeCycleActive
        AND NOT fbPatchDispense.IsBusy()
        AND NOT fbHeatStake.IsBusy()
        AND NOT fbVision.IsBusy()
        AND NOT stIndexStatus.bBusy
        AND (
            (bManualSupportTargetUpAtRejectStop
                AND stInputs.bStation2SupportExtended)
            OR
            ((NOT bManualSupportTargetUpAtRejectStop)
                AND stInputs.bStation2SupportRetracted)
        );

    IF bRejectChuteStopRequestLatched THEN
        IF bManualRejectStopReady THEN
            eMachineState := E_MachineState.Stopping;
        END_IF

    // Existing operator Stop behaviour remains unchanged.
    ELSIF stCommand.bStop OR stInputs.bEventCycleStopRequest THEN
        eMachineState := E_MachineState.Stopping;
    END_IF

E_MachineState.Fault:
    bAutoCycleStopRequestLatched := FALSE;

    // Immediate Fault always removes the pneumatic-supply memory.
    // Therefore Fault -> Reset -> Stopping -> Stopped remains depressurised
    // until a NEW System Initialising sequence explicitly turns air back on.
    bAirSupplyLatched := FALSE;
    stOutputsInternal.bAirSupplyEnable := FALSE;

    tonInitialising(IN := FALSE);
    tonStopping(IN := FALSE);

    // Latch Reset. PRG_Events runs after PRG_Main and may only clear
    // GVL_MASTER.bMachineFault later in this PLC scan. Without this latch,
    // a one-scan Reset pulse is lost before the machine can leave Fault.
    IF stCommand.bReset AND NOT bOutHMI THEN
        bFaultResetRequested := TRUE;
        bInitialisationTimeoutFault := FALSE;
        bStoppingTimeoutFault := FALSE;
        fbIndex.Reset();
    END_IF
	
		// Do not retain a pending Reset while HMI is unavailable.
	IF bOutHMI THEN
		bFaultResetRequested := FALSE;
	END_IF

    // Leave Fault only after Safety and the event system have both recovered.
    IF bFaultResetRequested
        AND stInputs.stSafety.bSafetyOk
        AND NOT stInputs.bEventFault
        AND NOT fbIndex.IsFaulted()
        AND NOT fbMainDoorLock.IsFaulted()
    THEN
        bFaultResetRequested := FALSE;
        eMachineState := E_MachineState.Stopping;
    END_IF
END_CASE

// Do not queue a rejected start behind HOME or a reserved image position.
// The raw two-hand edge was already sampled before Vision admission this scan.
bManualIndexBlockVision := NOT stVisionStatus.bHome
    OR fbVisionManualImages.bActive OR bVisionImageOwnedBeforeUpdate
    OR bVisionImageJogBusy OR bVisionManualHomeActive OR bVisionManualSequenceActive
    OR bVisionImageRecoveryRequired OR fbVisionManualImages.bFault OR bManualCameraRecoveryActive;
bManualIndexBlockHeat := NOT bHeatStakeManualHomePosition OR fbHeatStake.IsBusy();
bManualIndexBlockPatch := NOT bPatchVerticalIndexReady
    OR NOT (GVL_Motion.stPatchFeedSettings.bUsePatchVerticalFeedback OR stOutputsInternal.bPatchVerticalUp)
    OR fbPatchDispense.IsBusy() OR fbPatchFeedManager.stStatus.bDriveBusy
    OR bPatchManualVerticalDownHeld OR stOutputsInternal.bPatchVerticalDown;
bManualIndexBlockOther := NOT stInputs.stSafety.bMotionSafetyPermitted
    OR NOT stInputs.bMainDoorClosed OR NOT GVL_Safety.bAirSupplySafe
    OR bRejectChuteStopRequestLatched OR stCommand.bStop OR stCommand.bReset
    OR NOT stInputs.bIndexReady OR NOT stInputs.bIndexLocked
    OR (stInputs.eIndexPosition = E_TablePosition.Unknown)
    OR (fbIndex.GetState() <> E_IndexState.Idle) OR stIndexStatus.bTwoHandRequired;
bManualIndexStartAllowed := NOT bManualIndexBlockVision AND NOT bManualIndexBlockHeat
    AND NOT bManualIndexBlockPatch AND NOT bManualIndexBlockOther
    AND stPermissives.bIndexMoveAllowed;
IF bManualIndexAttempt THEN
    IF bManualIndexStartAllowed THEN
        bIndexMoveAccepted := fbIndex.RequestManualMove();
    ELSE
        bManualIndexWarningActive := TRUE;
    END_IF
END_IF
IF (eMachineState <> E_MachineState.Manual) OR bManualIndexStartAllowed THEN
    bManualIndexWarningActive := FALSE;
END_IF
GVL_MASTER.bManualIndexBlockVision := bManualIndexWarningActive AND bManualIndexBlockVision;
GVL_MASTER.bManualIndexBlockHeat := bManualIndexWarningActive AND bManualIndexBlockHeat;
GVL_MASTER.bManualIndexBlockPatch := bManualIndexWarningActive AND bManualIndexBlockPatch;
GVL_MASTER.bManualIndexBlockOther := bManualIndexWarningActive AND bManualIndexBlockOther;
IF NOT stVisionStatus.bHome THEN
    GVL_MASTER.sManualIndexVisionReason := 'Index blocked: Vision not HOME';
ELSIF bVisionImageJogBusy OR bVisionManualHomeActive OR bVisionManualSequenceActive THEN
    GVL_MASTER.sManualIndexVisionReason := 'Index blocked: Vision manual action active';
ELSIF bManualCameraRecoveryActive THEN
    GVL_MASTER.sManualIndexVisionReason := 'Index blocked: camera recovery in progress';
ELSIF fbVisionManualImages.bActive OR bVisionImageOwnedBeforeUpdate THEN
    GVL_MASTER.sManualIndexVisionReason := 'Index blocked: Vision position reserved';
ELSE
    GVL_MASTER.sManualIndexVisionReason := 'Index blocked: Vision recovery required';
END_IF
IF NOT stInputs.stSafety.bMotionSafetyPermitted THEN
    GVL_MASTER.sManualIndexOtherReason := 'Index blocked: motion safety not ready';
ELSIF NOT stInputs.bMainDoorClosed OR NOT GVL_Safety.bAirSupplySafe THEN
    GVL_MASTER.sManualIndexOtherReason := 'Index blocked: door or air not ready';
ELSIF bRejectChuteStopRequestLatched OR stCommand.bStop OR stCommand.bReset THEN
    GVL_MASTER.sManualIndexOtherReason := 'Index blocked: Stop/Reset request active';
ELSIF stInputs.eIndexPosition = E_TablePosition.Unknown THEN
    GVL_MASTER.sManualIndexOtherReason := 'Index blocked: position unknown';
ELSE
    GVL_MASTER.sManualIndexOtherReason := 'Index blocked: table not locked/idle or request pending';
END_IF

fbIndex.Cyclic(bEnable := (eMachineState <> E_MachineState.PowerUp) AND (eMachineState <> E_MachineState.Fault), bReset := stCommand.bReset, bAutomaticMode := (eMachineState = E_MachineState.AutoCycle), bManualMode := (eMachineState = E_MachineState.Manual), bMovePermissive := stPermissives.bIndexMoveAllowed, bSafetyMotionPermitted := stInputs.stSafety.bMotionSafetyPermitted, bTwoHandsSafe := stInputs.bTwoHandsSafe, bStationsHome := stPermissives.bStationsHome, bProcessToolingRetracted := stPermissives.bStationsIndexPermissive, bTableReady := stInputs.bIndexReady, bTableLocked := stInputs.bIndexLocked, bCompletedSensor := stInputs.bIndexCompletedSensor, bSupportExtended := TRUE, bSupportRetracted := TRUE, eCurrentPosition := stInputs.eIndexPosition, tRotateDelay := stConfig.tIndexRotateDelay, tStopDelay := stConfig.tIndexStopDelay, tSupportTimeout := stConfig.tIndexSupportTimeout, tMovementTimeout := stConfig.tIndexTimeout, tTwoHandHold := stConfig.tTwoHandHold, tTwoHandRecoveryTimeout := stConfig.tTwoHandRecoveryTimeout, bRotatePortA => stOutputsInternal.bIndexRotatePortA, bStopPortB => stOutputsInternal.bIndexStopPortB, bSupportExtendRequest => stOutputsInternal.bIndexSupportExtend, bSupportRetractRequest => stOutputsInternal.bIndexSupportRetract);
stIndexStatus := fbIndex.GetStatus();



///////////////////////////////////////////////////////////////////


// Use the state after the machine CASE transitions in this scan.
// Stopped -> Initialising must not drop an existing hot-door lock request.
// Same strategy as the validated Silicone Station.
// Door locking is requested independently from door feedback while the
// machine is in an active state that requires the door secured.
bAirAndDoorEnable :=
    (eMachineState = E_MachineState.Initialising)
    OR (eMachineState = E_MachineState.ReadyToStart)
    OR (eMachineState = E_MachineState.AutoCycle)
    OR (eMachineState = E_MachineState.Manual)
	OR (eMachineState = E_MachineState.Dwell);

 // =====================================================
 // MAIN DOOR - HOT TEMPERATURE PROTECTION
 // =====================================================

 // Reset acknowledgement when leaving Stopped.
 IF eMachineState <> E_MachineState.Stopped THEN
     bMainDoorUnlockAcknowledged := FALSE;

 // Accept acknowledgement only in Stopped.
 ELSIF GVL_HMI.stCommands.bManualMainDoorUnlock THEN
     bMainDoorUnlockAcknowledged := TRUE;
 END_IF;

 // Consume HMI command.
 GVL_HMI.stCommands.bManualMainDoorUnlock := FALSE;

 // Keep door locked in Stopped while heaters are hot,
 // until operator acknowledges.
 bMainDoorHotLockRequired :=
     (eMachineState = E_MachineState.Stopped)
     AND NOT bMainDoorUnlockAcknowledged
     // TC3 is head/body feedback; TC1/TC2 cartridge temperatures do not set this demand.
     // Equality requires acknowledgement; an unordered/NaN value is not considered cool.
     AND NOT (stHeatStakeTemperatureStatus.rOverTempTemperatureC <
         GVL_Config.rMainDoorHotTemperatureLimitC);

 // =====================================================
 // MAIN DOOR SUPERVISION
 // =====================================================

 fbMainDoorLock.Cyclic(
     // Supervise the same lock demand sent to TwinSAFE, including hot-door retention.
     // Retain an existing lock through the entry scan: feeder stop permissions
     // take effect next scan. Never create a new lock demand on PowerUp/recovery.
     bEnableAutomatic := bAirAndDoorEnable
         OR ((eMachineState = E_MachineState.Stopping)
             AND (((ePreviousMachineState <> E_MachineState.Stopping)
                     AND stMainDoorStatus.bLockRequest)
                 OR fbPatchFeedManager.stStatus.bBusy))
         OR bMainDoorHotLockRequired,
     bManualEnable := FALSE,
     bManualLockRequest := FALSE,
     bManualUnlockRequest := FALSE,

     bStopRequest :=
         (eMachineState = E_MachineState.Fault)
         OR ((eMachineState = E_MachineState.Stopping)
             AND (ePreviousMachineState = E_MachineState.Stopping)
             AND NOT fbPatchFeedManager.stStatus.bBusy)
         OR (
             (eMachineState = E_MachineState.Stopped)
             AND NOT bMainDoorHotLockRequired
         ),

     bResetRequest := stCommand.bReset,
     bDoorClosed := stInputs.bMainDoorClosed,
     bDoorLocked := stInputs.bMainDoorLocked,
     bIndexBusy := stIndexStatus.bBusy,
     bProcessSafePosition := NOT fbPatchFeedManager.stStatus.bBusy,
     tLockTimeout := stConfig.tDoorLockTimeout,
     tUnlockTimeout := stConfig.tDoorUnlockTimeout,
     bDoorUnsafe := stInputs.bMainDoorUnsafe,
     bLockOutput => bDoorLockOutput
 );

 stMainDoorStatus := fbMainDoorLock.GetStatus();

 // =====================================================
 // PHYSICAL DOOR LOCK REQUEST
 // =====================================================

 stOutputsInternal.bMainDoorLockRequest :=
     bAirAndDoorEnable
     OR ((eMachineState = E_MachineState.Stopping)
             AND (((ePreviousMachineState <> E_MachineState.Stopping)
                     AND stMainDoorStatus.bLockRequest)
                 OR fbPatchFeedManager.stStatus.bBusy))
     OR bMainDoorHotLockRequired;

	///////////////////////////////

// Re-check after component cyclic execution so a fault detected in this scan
// drops TwinSAFE immediately rather than waiting for the following PLC scan.
// Existing event/process-cycle faults are allowed during Initialising so the
// machine can restore pneumatic tooling to HOME.
IF (
        stInputs.bEventFault
        AND (eMachineState <> E_MachineState.Initialising)
    )
    OR fbIndex.IsFaulted()
    OR fbMainDoorLock.IsFaulted()
    OR (
        bProcessCycleFault
        AND (eMachineState <> E_MachineState.Initialising)
    )
    OR stHeatStakeTemperatureStatus.bFault
    OR bInitialisationTimeoutFault
    OR bStoppingTimeoutFault
	OR bHeaterDwellTimeoutFault
THEN
    bSafetyDropRequest := TRUE;
    eMachineState := E_MachineState.Fault;
END_IF

// Finalise the affected parts before automatic operation resumes.
IF (eMachineState = E_MachineState.Fault)
    AND (ePreviousMachineState = E_MachineState.AutoCycle)
THEN
    stProcessFaultResult.bValid := TRUE;
    stProcessFaultResult.bPassed := FALSE;
    stProcessFaultResult.eCode := E_ProcessResultCode.Aborted;
    stProcessFaultResult.udiFaultCode := 0;
    stProcessFaultResult.udiAlertCode := 0;

    stPatchDispenseNest := fbNestManager.GetNestAtPosition(stConfig.ePatchDispensePosition);
    stHeatStakeNest := fbNestManager.GetNestAtPosition(stConfig.eHeatStakePosition);
    stVisionNest := fbNestManager.GetNestAtPosition(stConfig.eVisionPosition);

    IF bPatchDispenseRequired AND (stPatchDispenseNest.ePatchDispenseStage = E_NestStageStatus.Waiting) THEN
        stProcessFaultResult.sDetail := 'Patch Dispense incomplete - Reject';
        fbNestManager.StorePatchDispenseResultAtPosition(stConfig.ePatchDispensePosition, stProcessFaultResult);
        FinaliseAndRecordAtPosition(stConfig.ePatchDispensePosition);
    END_IF

    IF bHeatStakeRequired AND (stHeatStakeNest.eHeatStakeStage = E_NestStageStatus.Waiting) THEN
        stProcessFaultResult.sDetail := 'Heat Stake interrupted - Reject';
        fbNestManager.StoreHeatStakeResultAtPosition(stConfig.eHeatStakePosition, stProcessFaultResult);
        FinaliseAndRecordAtPosition(stConfig.eHeatStakePosition);
    END_IF

    IF stVisionNest.bPartPresent
        AND (stVisionNest.eVisionStage = E_NestStageStatus.Waiting)
        AND (bVisionProcessingBeforeUpdate
            OR (bVisionRequired AND fbVision.IsFaulted()))
    THEN
        stProcessFaultResult.sDetail := 'Vision interrupted - Reject';
        fbNestManager.StoreVisionResultAtPosition(stConfig.eVisionPosition, stProcessFaultResult);
        FinaliseAndRecordAtPosition(stConfig.eVisionPosition);
    END_IF
END_IF

// Validated Silicone-station handshake:
// - Run/Stop is normally TRUE so TwinSAFE is running and can return Safety_OK.
// - A PLC-originated immediate fault pulses Run/Stop FALSE for 500 ms.
// - It then returns TRUE automatically, even while the machine remains in Fault,
//   allowing TwinSAFE to recover and Safety_OK to become TRUE for operator Reset.
tpSafetyRunDrop(
    IN := bSafetyDropRequest,
    PT := T#500MS
);

stOutputsInternal.bSafetyRunRequest := NOT tpSafetyRunDrop.Q;

stOutputsInternal.bSafetyResetRequest := stCommand.bReset AND NOT stInputs.stSafety.bSafetyOk;
stOutputsInternal.bSafetyErrorAcknowledgementRequest := stOutputsInternal.bSafetyResetRequest;
// =========================================================
// OPERATOR LIGHTS - SILICONE STATION BEHAVIOUR
// =========================================================
// Start flashes only while ReadyToStart.
stOutputsInternal.bLedStart :=
    (eMachineState = E_MachineState.ReadyToStart)
    AND bLedBlinkState;

// Reset flashes while operator Reset is expected.
stOutputsInternal.bLedReset :=
    (
        (eMachineState = E_MachineState.PowerUp)
        OR (eMachineState = E_MachineState.Fault)
        OR (eMachineState = E_MachineState.Stopped)
    )
    AND bLedBlinkState;

// -------------------------------------------------------------------------
// Operator PASS / FAIL result lights
// -------------------------------------------------------------------------
// Customer-agreed behaviour:
// - both lights are OFF by default;
// - machine Fault must NEVER use the FAIL/result light;
// - lights are used only in AutoCycle;
// - a valid PASS/FAIL result must exist at the operator nest;
// - the physical part must still be present at the loading/operator nest;
// - immediately after the operator removes the part, both lights turn OFF.
//
// Result-record clearing can occur later as part of the normal operator/reject
// workflow. The physical presence condition intentionally makes the lamp go
// dark immediately on part removal, independent of when the nest result is
// finally cleared.
IF (eMachineState = E_MachineState.AutoCycle)
    AND stOperatorNest.stResult.bValid
    AND stInputs.bLoadingStationEaglePresent
THEN
    stOutputsInternal.bLedPass := stOperatorNest.stResult.bPassed;
    stOutputsInternal.bLedFail := NOT stOperatorNest.stResult.bPassed;
ELSE
    stOutputsInternal.bLedPass := FALSE;
    stOutputsInternal.bLedFail := FALSE;
END_IF

// Lighting:
// - Internal machine light is on while the main door is open.
// - Operator/nest light is controlled by the Main-screen LIGHT toggle.
stOutputsInternal.bInternalLight := NOT stInputs.bMainDoorClosed;
stOutputsInternal.bNestLight := stCommand.bOperatorLight;
// -------------------------------------------------------------------------
// Heat Stake HMI status - Manual Mode tooling position
// -------------------------------------------------------------------------
// Keep the station FB free of Manual Mode oscillation, but present BUSY to the
// engineer whenever the tooling is not in its complete home position.
//
// This deliberately does NOT feed back into the individual recovery-button
// permissives. Otherwise, for example, extending the support would make Busy
// TRUE and disable the same toggle needed to retract it again.
IF eMachineState = E_MachineState.Manual THEN
    stHeatStakeStatus.bBusy :=
        fbHeatStake.IsBusy()
        OR (usiHeatStakeManualActionStep <> 0)
        OR NOT (
            stInputs.bStation2SupportRetracted
            AND stInputs.bHeatStakeHeadUp
            AND NOT stInputs.bHeatStakeHeadDown
            AND NOT bHeatStakeManualHeadUnlocked
        );

    // A station that is manually out of HOME is not operationally Ready.
    stHeatStakeStatus.bReady :=
        stHeatStakeStatus.bReady
        AND NOT stHeatStakeStatus.bBusy;
END_IF

// Single-solenoid head valve: retain the requested direction between legacy pulses.
// Reservoir air and maintained valve power are required for physical fault retraction.
IF NOT stInputs.stSafety.bSafetyOk
    OR NOT stInputs.stSafety.bProcessSafetyPermitted
    OR NOT GVL_Safety.bAirSupplySafe
    OR (eMachineState = E_MachineState.Fault) THEN
    bHeatStakeHeadUpRecoveryLatched := TRUE;
    bHeatStakeHeadDownHeld := FALSE;
ELSIF (ePreviousMachineState = E_MachineState.Initialising)
    AND (eMachineState = E_MachineState.ReadyToStart)
    AND stInputs.bHeatStakeHeadUp
    AND NOT stInputs.bHeatStakeHeadDown THEN
    // Reset/safety recovery alone must never re-arm descent.
    bHeatStakeHeadUpRecoveryLatched := FALSE;
    bHeatStakeHeadDownHeld := FALSE;
END_IF

IF bHeatStakeHeadUpRecoveryLatched OR bHeatStakeHeadUpRequest THEN
    bHeatStakeHeadDownHeld := FALSE; // UP wins conflicting requests.
ELSIF bHeatStakeHeadDownRequest THEN
    bHeatStakeHeadDownHeld := TRUE;
END_IF

stOutputsInternal.bHeatStakeHeadDown := bHeatStakeHeadDownHeld
    AND NOT bHeatStakeHeadUpRecoveryLatched;
stOutputsInternal.bHeatStakeHeadUp := NOT stOutputsInternal.bHeatStakeHeadDown;

// Maintain Down Pressure for the complete retained DOWN command, including
// the manual hold after DOWN feedback ends the movement action.
// Evaluate after final direction/recovery arbitration so UP removes pressure
// in the same scan. Keep the regulator's existing limits and scaling.
rHeatStakePressureCommandBar := stHeatStakeProcessSettings.rDownPressureBar;
fbHeatStakePressureRegulator.Cyclic(
    bEnable := stOutputsInternal.bHeatStakeHeadDown,
    rSetpointBar := rHeatStakePressureCommandBar,
    rCommandBar => rHeatStakePressureScaledBar,
    iOutputRaw => iHeatStakePressureRaw
);
stOutputsInternal.iHeatStakePressureRaw := iHeatStakePressureRaw;
stHeatStakeProcessStatus.rPressureCommandBar := rHeatStakePressureScaledBar;
stHeatStakeProcessStatus.iPressureOutputRaw := iHeatStakePressureRaw;

stOutputs := stOutputsInternal;
stStatus.eMachineState := eMachineState;
stStatus.eProcessCycleState := eProcessCycleState;
stStatus.eIndexState := fbIndex.GetState();
stStatus.stIndexStatus := stIndexStatus;
stStatus.stMainDoorLock := stMainDoorStatus;
stStatus.eInitialisingWaitReason := eInitialisingWaitReason;
stStatus.eStoppingWaitReason := eStoppingWaitReason;
stStatus.eOperatorExchangeState := fbOperatorStation.GetState();
stStatus.eOperatorInstruction := fbOperatorStation.GetInstruction();
stStatus.stOperatorStation := stOperatorStatus;
stStatus.stPatchDispense := stPatchDispenseStatus;
stStatus.stHeatStake := stHeatStakeStatus;
stStatus.stHeatStakeTemperature := stHeatStakeTemperatureStatus;
stStatus.stHeatStakeProcess := stHeatStakeProcessStatus;
stStatus.bHeatStakeManualEnableAllowed := bHeatStakeManualEnableAllowed;
stStatus.bHeatStakeManualStakeAllowed := bHeatStakeManualStakeAllowed;
stStatus.bHeatStakeManualUnlockAllowed := bHeatStakeManualUnlockAllowed;
stStatus.bHeatStakeManualLockAllowed := bHeatStakeManualLockAllowed;
stStatus.bHeatStakeManualHeadDownAllowed := bHeatStakeManualHeadDownAllowed;
stStatus.bHeatStakeManualHeadUpAllowed := bHeatStakeManualHeadUpAllowed;
stStatus.bHeatStakeManualSupportAllowed := bHeatStakeManualSupportAllowed;
stStatus.bHeatStakeManualActionBusy := bHeatStakeManualActionBusy;
stStatus.bHeatStakeManualHeadUnlocked := bHeatStakeManualHeadUnlocked;
stStatus.stVision := stVisionStatus;
// Manual image presentation uses its actual owner, not the disabled automatic FB.
// Physical HOME and all automatic result/stage semantics remain unchanged.
IF (eMachineState = E_MachineState.Manual) AND stCommand.bVisionManualEnable
    AND NOT bVisionManualSequenceActive AND NOT bVisionManualHomeActive THEN
    stStatus.stVision.bBusy := GVL_HMI.bCameraManualBusy;
    stStatus.stVision.bFault := stVisionStatus.bFault OR fbVisionManualImages.bFault;
    // Station HOME is ready before Prepare; capture readiness remains a separate status.
    stStatus.stVision.bReady := (stVisionStatus.bHome OR fbVisionManualImages.bPrepared)
        AND stVisionStatus.bCommissioned AND stInputs.stSafety.bSafetyOk
        AND GVL_Safety.bAirSupplySafe AND NOT GVL_HMI.bCameraManualBusy
        AND NOT stStatus.stVision.bFault;
    stStatus.stVision.sDiagnostic := GVL_HMI.sCameraManualMessage;
END_IF
stStatus.bReady := (eMachineState = E_MachineState.ReadyToStart);
stStatus.bBusy := (eMachineState = E_MachineState.AutoCycle) OR stIndexStatus.bBusy;
stStatus.bFaulted := (eMachineState = E_MachineState.Fault);
stStatus.bInitialisationTimeoutFault := bInitialisationTimeoutFault;
stStatus.bStoppingTimeoutFault := bStoppingTimeoutFault;
stStatus.bProcessCycleTimeoutFault := bProcessCycleTimeoutFault;
stStatus.bSafetyStopRequested := tpSafetyRunDrop.Q;
stStatus.bSafetyRunRequested := stOutputsInternal.bSafetyRunRequest;
stStatus.bEventFault := stInputs.bEventFault;
stStatus.bCycleStopRequested := stInputs.bEventCycleStopRequest;
stStatus.bIndexPermissive := stPermissives.bIndexMoveAllowed;
stStatus.bEnableSetting := (eMachineState = E_MachineState.Stopped);
stStatus.bAllStationsCommissioned := bPatchDispenseCommissioned AND bHeatStakeCommissioned AND bVisionCommissioned;
stStatus.bAutoCycleAllowed := bAutoCycleAllowed;
stStatus.bDisabledNestPartIndexBlocked := bDisabledNestPartPresent;
stStatus.bDisabledNestPartPopupRequest := bDisabledNestPartPopupRequest;
stStatus.uiDisabledNestPartPopupNestId := uiDisabledNestPartPopupNestId;
stStatus.bRejectChuteFullLatched := bRejectChuteFullLatched;
stStatus.bRejectChutePopupRequest := bRejectChutePopupRequest;
stStatus.bRejectChuteStopRequest := bRejectChuteStopRequestLatched;
stStatus.bRejectChuteResetBlocked := bRejectChuteFullLatched;
stStatus.bHeatStakeHeadUp := stInputs.bHeatStakeHeadUp;
stStatus.bHeatStakeHeadDown := stInputs.bHeatStakeHeadDown;
stStatus.bHeatStakeHeadDownTimeoutFault := bHeatStakeStationHeadDownTimeoutFault OR bHeatStakeManualHeadDownTimeoutFault;
stStatus.bHeatStakeHeadUpTimeoutFault := bHeatStakeStationHeadUpTimeoutFault OR bHeatStakeManualHeadUpTimeoutFault;
stStatus.bHeatStakeHeadSensorConflictFault := bHeatStakeStationHeadSensorConflictFault OR (stInputs.bHeatStakeHeadUp AND stInputs.bHeatStakeHeadDown);
stStatus.stPermissives := stPermissives;
// Refresh published records after same-scan admission/reject updates.
aNestSnapshot := fbNestManager.GetAllNests();
stStatus.aNest := aNestSnapshot;
stStatus.aNestStatistics := fbNestManager.GetAllNestStatistics();
stStatus.sAutoCycleBlockReason := sAutoCycleBlockReason;
stStatus.sOperatorMessage := stOperatorStatus.sMessage;
stStatus.bHeaterDwellTimeoutFault := bHeaterDwellTimeoutFault;


// =====================================================
// VISION MANUAL MODE - HMI STATUS
// =====================================================
stStatus.bVisionManualEnableAllowed := bVisionManualEnableAllowed;
IF fbVisionManualImages.bActive OR fbVisionManualImages.bFault THEN
    bVisionHorizontalBackAllowed := FALSE;
    bVisionHorizontalFrontAllowed := FALSE;
    bVisionVerticalUpAllowed := FALSE;
    bVisionVerticalFullDownAllowed := FALSE;
    bVisionGripOpenAllowed := FALSE;
    bVisionGripCloseAllowed := FALSE;
    bVisionRotate0Allowed := FALSE;
    bVisionRotate180Allowed := FALSE;
END_IF
stStatus.bVisionManualRunSequenceAllowed :=bVisionManualRunSequenceAllowed;

stStatus.bVisionManualHomeAllowed := bVisionManualHomeAllowed;

// Vision physical HOME position.
stStatus.bVisionHome :=
    stInputs.bHorizontalMiniSlideExtended
    AND NOT stInputs.bHorizontalMiniSlideRetracted
    AND stInputs.bVerticalMiniSlideRetracted
    AND NOT stInputs.bVerticalMiniSlideExtended
    AND stInputs.bRotaryGripperOpened
    AND NOT stInputs.bRotaryGripperClosed
    AND bVisionRotate0Confirmed
    AND NOT bVisionRotate180Confirmed;
	


stStatus.bVisionHorizontalBackAllowed := bVisionHorizontalBackAllowed;
stStatus.bVisionHorizontalFrontAllowed := bVisionHorizontalFrontAllowed;

stStatus.bVisionVerticalUpAllowed := bVisionVerticalUpAllowed;
stStatus.bVisionVerticalIntermediateAllowed := FALSE; // Retired compatibility field.
stStatus.bVisionVerticalFullDownAllowed := bVisionVerticalFullDownAllowed;

stStatus.bVisionGripOpenAllowed := bVisionGripOpenAllowed;
stStatus.bVisionGripCloseAllowed := bVisionGripCloseAllowed;

stStatus.bVisionRotate0Allowed := bVisionRotate0Allowed;
stStatus.bVisionRotate180Allowed := bVisionRotate180Allowed;

stStatus.bVisionSupportAllowed := FALSE; // Retired compatibility field.

// Physical feedback for HMI LEDs.
stStatus.bVisionHorizontalBack := stInputs.bHorizontalMiniSlideExtended;
stStatus.bVisionHorizontalFront := stInputs.bHorizontalMiniSlideRetracted;

stStatus.bVisionVerticalUp := stInputs.bVerticalMiniSlideRetracted;
stStatus.bVisionVerticalDown := stInputs.bVerticalMiniSlideExtended;

stStatus.bVisionGripOpen := stInputs.bRotaryGripperOpened;
stStatus.bVisionGripClosed := stInputs.bRotaryGripperClosed;

stStatus.bVisionRotate0 := bVisionRotate0Confirmed;
stStatus.bVisionRotate180 := bVisionRotate180Confirmed;

stStatus.bVisionSupportExtended := FALSE; // Retired compatibility field.
stStatus.bVisionSupportRetracted := FALSE; // Retired compatibility field.

CASE eMachineState OF
    E_MachineState.PowerUp:
        stStatus.sMachineMessage := 'System power up';

    E_MachineState.Initialising:
        stStatus.sMachineMessage := 'System initialising';

    E_MachineState.ReadyToStart:
        IF stHeatStakeTemperatureStatus.bLowTemperature THEN
            stStatus.sMachineMessage := 'Heat Stake preheating';
        ELSIF bAutoCycleAllowed THEN
            stStatus.sMachineMessage := 'System ready to start';
        ELSE
            stStatus.sMachineMessage := sAutoCycleBlockReason;
        END_IF
    E_MachineState.Dwell:

		
// Convert live temperature values to text.
sHeaterMinimum := LREAL_TO_STRING(
    GVL_MASTER.stStatus.stHeatStakeTemperature.rLowLimitC
);

sHeaterCurrent := LREAL_TO_STRING(
    GVL_MASTER.stStatus.stHeatStakeTemperature.rOverTempTemperatureC
);

        stStatus.sMachineMessage := 
			CONCAT(CONCAT(CONCAT(CONCAT(' Heater Temp below Limit: ',sHeaterMinimum),' Â°C | Current Temp: '),sHeaterCurrent),' Â°C ') ;

    E_MachineState.AutoCycle:
        // Operator message priority:
        //
        // 1. While any process station is active, show one generic process
        //    message rather than the operator-exchange text.
        // 2. Failed/passed-part removal and reject instructions retain
        //    priority once processing is finished.
        // 3. When the cycle has returned to the normal index-wait state,
        //    explicitly tell the operator the machine is ready to index.
        // 4. Fall back to the current OperatorStation message.

        IF stHeatStakeTemperatureStatus.bLowTemperature
            AND NOT stHeatStakeTemperatureStatus.bFault
        THEN
            stStatus.sMachineMessage := 'Heat Stake warming up - index inhibited';

        ELSIF bAnyStationInProcess THEN
            stStatus.sMachineMessage := 'In process';

        ELSIF
            (stOperatorStatus.eState = E_OperatorExchangeState.WaitingForPartRemoval)
            OR (stOperatorStatus.eState = E_OperatorExchangeState.WaitingForRejectConfirmation)
        THEN
            stStatus.sMachineMessage := stOperatorStatus.sMessage;

        ELSIF eProcessCycleState = E_CycleState.WaitingForProcessCycleTrigger THEN
            stStatus.sMachineMessage := 'Ready for index - press touch buttons';

        ELSIF LEN(stOperatorStatus.sMessage) > 0 THEN
            stStatus.sMachineMessage := stOperatorStatus.sMessage;

        ELSE
            stStatus.sMachineMessage := 'System auto cycle';
        END_IF

    E_MachineState.Manual:
        stStatus.sMachineMessage := 'Manual mode';

    E_MachineState.Stopping:
        stStatus.sMachineMessage := 'Stopping';

    E_MachineState.Stopped:
        stStatus.sMachineMessage := 'Cycle stopped';

    E_MachineState.Fault:
        stStatus.sMachineMessage := 'Immediate fault';
END_CASE

IF bRejectChuteFullLatched
    AND (eMachineState <> E_MachineState.Fault)
THEN
    stStatus.sMachineMessage :=
        'Reject chute full - empty chute and press Acknowledge';
END_IF

// Must be the final machine-state assignment in Cyclic.
// Used on the next scan to detect one-shot transitions into Fault.
ePreviousMachineState := eMachineState;

// Track FINAL published outputs, after all machine fault/output overrides.
bPatchVerticalUpCommandPrevious := stOutputs.bPatchVerticalUp;
bPatchVerticalDownCommandPrevious := stOutputs.bPatchVerticalDown;

// Track final commands after all fault/output overrides.
bVisionRotate0CommandPrevious := stOutputs.bVisionRotate0;
bVisionRotate180CommandPrevious := stOutputs.bVisionRotate180;
END_METHOD

METHOD PRIVATE FinaliseAndRecordAtPosition
VAR_INPUT
    ePosition : E_TablePosition;
END_VAR
VAR
    stHistoryNest : ST_Nest;
    stCSVRecord : ST_CycleDataCSV;
END_VAR
stHistoryNest := fbNestManager.GetNestAtPosition(ePosition);
IF NOT stHistoryNest.bPartPresent OR stHistoryNest.bStatisticsCounted THEN
    RETURN;
END_IF

IF fbNestManager.FinaliseResultAtPosition(ePosition) THEN
    stHistoryNest := fbNestManager.GetNestAtPosition(ePosition);
    // =================================================
    // TEST HISTORY
    // =================================================

    IF stHistoryNest.bPartPresent
        AND stHistoryNest.stResult.bValid
    THEN

        // ---------------------------------------------
        // GENERAL RESULT
        // ---------------------------------------------

        GVL_Persistent.astTestHistory[
            GVL_Persistent.uiTestHistoryWriteIndex
        ].uiNestId := stHistoryNest.nId;

        GVL_Persistent.astTestHistory[
            GVL_Persistent.uiTestHistoryWriteIndex
        ].eResult := stHistoryNest.eDisposition;


        // ---------------------------------------------
        // PATCH DISPENSE
        // ---------------------------------------------

        GVL_Persistent.astTestHistory[
            GVL_Persistent.uiTestHistoryWriteIndex
        ].bPatchDispenseValid :=
            stHistoryNest.stPatchDispenseResult.bValid;

        GVL_Persistent.astTestHistory[
            GVL_Persistent.uiTestHistoryWriteIndex
        ].bPatchDispensePass :=
            stHistoryNest.stPatchDispenseResult.bPassed;


        // ---------------------------------------------
        // HEAT STAKE
        // ---------------------------------------------

        GVL_Persistent.astTestHistory[
            GVL_Persistent.uiTestHistoryWriteIndex
        ].bHeatStakeValid :=
            stHistoryNest.stHeatStakeResult.bValid;

        GVL_Persistent.astTestHistory[
            GVL_Persistent.uiTestHistoryWriteIndex
        ].bHeatStakePass :=
            stHistoryNest.stHeatStakeResult.bPassed;


        // ---------------------------------------------
        // VISION
        // ---------------------------------------------

        GVL_Persistent.astTestHistory[
            GVL_Persistent.uiTestHistoryWriteIndex
        ].bVisionValid :=
            stHistoryNest.stVisionResult.bValid;

        GVL_Persistent.astTestHistory[
            GVL_Persistent.uiTestHistoryWriteIndex
        ].bVisionPass :=
            stHistoryNest.stVisionResult.bPassed;

		// Store individual Vision inspection results
		// for persistent history and future CSV integration.

		GVL_Persistent.astTestHistory[
			GVL_Persistent.uiTestHistoryWriteIndex
		].stVisionInspectionResults :=
			stHistoryNest.stVisionResult.CameraResults;


        // ---------------------------------------------
        // DATE / TIME
        // ---------------------------------------------

        GVL_Persistent.astTestHistory[
            GVL_Persistent.uiTestHistoryWriteIndex
        ].sDate := GVL_MASTER.sSystemDate;

        GVL_Persistent.astTestHistory[
            GVL_Persistent.uiTestHistoryWriteIndex
        ].sTime := GVL_MASTER.sSystemTime;


        // ---------------------------------------------
        // FINAL RESULT TEXT
        // ---------------------------------------------

        IF stHistoryNest.stResult.bPassed THEN

            GVL_Persistent.astTestHistory[
                GVL_Persistent.uiTestHistoryWriteIndex
            ].sResult := 'PASS';

        ELSE

            GVL_Persistent.astTestHistory[
                GVL_Persistent.uiTestHistoryWriteIndex
            ].sResult := 'FAIL';

        END_IF;


        // ---------------------------------------------
        // PATCH DISPENSE RESULT TEXT
        // ---------------------------------------------

        IF NOT stHistoryNest.stPatchDispenseResult.bValid THEN

            GVL_Persistent.astTestHistory[
                GVL_Persistent.uiTestHistoryWriteIndex
            ].sPatchDispenseResult := 'NOT TESTED';

        ELSIF stHistoryNest.stPatchDispenseResult.bPassed THEN

            GVL_Persistent.astTestHistory[
                GVL_Persistent.uiTestHistoryWriteIndex
            ].sPatchDispenseResult := 'PASS';

        ELSE

            GVL_Persistent.astTestHistory[
                GVL_Persistent.uiTestHistoryWriteIndex
            ].sPatchDispenseResult := 'FAIL';

        END_IF;


        // ---------------------------------------------
        // HEAT STAKE RESULT TEXT
        // ---------------------------------------------

        IF NOT stHistoryNest.stHeatStakeResult.bValid THEN

            GVL_Persistent.astTestHistory[
                GVL_Persistent.uiTestHistoryWriteIndex
            ].sHeatStakeResult := 'NOT TESTED';

        ELSIF stHistoryNest.stHeatStakeResult.bPassed THEN

            GVL_Persistent.astTestHistory[
                GVL_Persistent.uiTestHistoryWriteIndex
            ].sHeatStakeResult := 'PASS';

        ELSE

            GVL_Persistent.astTestHistory[
                GVL_Persistent.uiTestHistoryWriteIndex
            ].sHeatStakeResult := 'FAIL';

        END_IF;


        // ---------------------------------------------
        // VISION RESULT TEXT
        // ---------------------------------------------

        IF NOT stHistoryNest.stVisionResult.bValid THEN

            GVL_Persistent.astTestHistory[
                GVL_Persistent.uiTestHistoryWriteIndex
            ].sVisionResult := 'NOT TESTED';

        ELSIF stHistoryNest.stVisionResult.bPassed THEN

            GVL_Persistent.astTestHistory[
                GVL_Persistent.uiTestHistoryWriteIndex
            ].sVisionResult := 'PASS';

        ELSE

            GVL_Persistent.astTestHistory[
                GVL_Persistent.uiTestHistoryWriteIndex
            ].sVisionResult := 'FAIL';

        END_IF;


        // Hand off the recorded result to the CSV writer in FIFO order.
        stCSVRecord.uiNestId := GVL_Persistent.astTestHistory[GVL_Persistent.uiTestHistoryWriteIndex].uiNestId;
        stCSVRecord.sGeneralResult := GVL_Persistent.astTestHistory[GVL_Persistent.uiTestHistoryWriteIndex].sResult;
        stCSVRecord.sPatchDispenseResult := GVL_Persistent.astTestHistory[GVL_Persistent.uiTestHistoryWriteIndex].sPatchDispenseResult;
        stCSVRecord.sHeatStakeResult := GVL_Persistent.astTestHistory[GVL_Persistent.uiTestHistoryWriteIndex].sHeatStakeResult;
        stCSVRecord.sVisionResult := GVL_Persistent.astTestHistory[GVL_Persistent.uiTestHistoryWriteIndex].sVisionResult;
        stCSVRecord.sDate := GVL_Persistent.astTestHistory[GVL_Persistent.uiTestHistoryWriteIndex].sDate;
        stCSVRecord.sTime := GVL_Persistent.astTestHistory[GVL_Persistent.uiTestHistoryWriteIndex].sTime;

        IF NOT GVL_Persistent.bCSVPendingRecord THEN
            GVL_Persistent.stCSVPendingRecord := stCSVRecord;
            GVL_Persistent.bCSVPendingRecord := TRUE;
        ELSIF GVL_Persistent.uiCSVAdditionalPendingCount < 2 THEN
            GVL_Persistent.aCSVAdditionalPendingRecords[GVL_Persistent.uiCSVAdditionalPendingCount] := stCSVRecord;
            GVL_Persistent.uiCSVAdditionalPendingCount := GVL_Persistent.uiCSVAdditionalPendingCount + 1;
        ELSE
            GVL_Persistent.udiCSVRecordsDropped := GVL_Persistent.udiCSVRecordsDropped + 1;
            GVL_Persistent.bCSVQueueOverflow := TRUE;
        END_IF

		// ---------------------------------------------
        // ADVANCE HISTORY BUFFER
        // ---------------------------------------------

        IF GVL_Persistent.uiTestHistoryCount < 2001 THEN

            GVL_Persistent.uiTestHistoryCount :=
                GVL_Persistent.uiTestHistoryCount + 1;

        END_IF;

        IF GVL_Persistent.uiTestHistoryWriteIndex < 2000 THEN

            GVL_Persistent.uiTestHistoryWriteIndex :=
                GVL_Persistent.uiTestHistoryWriteIndex + 1;

        ELSE

            GVL_Persistent.uiTestHistoryWriteIndex := 0;

        END_IF;

    END_IF;
END_IF
END_METHOD

METHOD PRIVATE ResetCyclicOutputs
stOutputsInternal.bSafetyRunRequest := FALSE;
stOutputsInternal.bSafetyResetRequest := FALSE;
stOutputsInternal.bSafetyErrorAcknowledgementRequest := FALSE;
stOutputsInternal.bAirSupplyEnable := FALSE;
stOutputsInternal.bMainDoorLockRequest := FALSE;
stOutputsInternal.bIndexRotatePortA := FALSE;
stOutputsInternal.bIndexStopPortB := FALSE;
stOutputsInternal.bIndexSupportExtend := FALSE;
stOutputsInternal.bIndexSupportRetract := FALSE;
stOutputsInternal.bStation1SupportExtend := FALSE;
stOutputsInternal.bStation1SupportRetract := FALSE;
stOutputsInternal.bStation2SupportExtend := FALSE;
stOutputsInternal.bStation2SupportRetract := FALSE;
stOutputsInternal.bStation3SupportExtend := FALSE;
stOutputsInternal.bStation3SupportRetract := FALSE;
stOutputsInternal.bVisionHorizontalBack := FALSE;
stOutputsInternal.bVisionHorizontalFront := FALSE;
stOutputsInternal.bVisionVerticalUp := FALSE;
stOutputsInternal.bVisionVerticalDown := FALSE;
stOutputsInternal.bVisionLimitOff := FALSE;
stOutputsInternal.bVisionLimitOn := FALSE;
stOutputsInternal.bVisionGripClose := FALSE;
stOutputsInternal.bVisionGripOpen := FALSE;
stOutputsInternal.bVisionRotate0 := FALSE;
stOutputsInternal.bVisionRotate180 := FALSE;
stOutputsInternal.bHeatStakeHeadLock := FALSE;
stOutputsInternal.bHeatStakeHeadUnlock := FALSE;
stOutputsInternal.bHeatStakeHeadDown := FALSE;
stOutputsInternal.bHeatStakeHeadUp := FALSE;
stOutputsInternal.iHeatStakePressureRaw := 0;
stOutputsInternal.bLedStart := FALSE;
stOutputsInternal.bLedReset := FALSE;
stOutputsInternal.bLedPass := FALSE;
stOutputsInternal.bLedFail := FALSE;
END_METHOD

END_FUNCTION_BLOCK

(* stored: Version 1.1.0.1, ProductVersion 3.1.4026.18
   POU FB_IndexedPatchPressMachine: Id {cd45b888-3938-49e7-a56e-6a78ef36b4a7}, SpecialFunc None
   Method Cyclic: Id {a779d1da-ccea-489e-9adf-3c1ac0c82903}
   Method FinaliseAndRecordAtPosition: Id {dbe17950-e44a-40e0-8569-211937468bbf}
   Method ResetCyclicOutputs: Id {2afcae24-43c4-4871-871e-9348e38cf5c0} *)
